FUNCTION F_vltSign : LREAL
VAR_INPUT
	number:	LREAL;
END_VAR
VAR
END_VAR

(*
static double vltSign(double number)
{
    if (number >= 0)
	return 1.0;
    return -1.0;
}
*)

IF number >= 0 THEN
	F_vltSign	:= 1.0;
ELSE
	F_vltSign	:= -1.0;
END_IF

END_FUNCTION

(* stored: Version 1.1.0.1, ProductVersion 3.1.4022.9
   POU F_vltSign: Id {465ce45f-8d25-42cb-bc38-eff9299e050f}, SpecialFunc None *)
